KUKA KRL data list: C3_getcube.dat

&ACCESS RVO
&REL 4
&PARAM DISKPATH = KRC:\R1\Program
DEFDAT  C3_getcube PUBLIC

DECL E6POS XP1={X 224.960861,Y 55.9276581,Z 35.7754402,A 162.906586,B 89.0492325,C -106.826286,S 2,T 10,E1 0.0,E2 0.0,E3 0.0,E4 0.0,E5 0.0,E6 0.0}
DECL FDAT FP1={TOOL_NO 14,BASE_NO 2,IPO_FRAME #BASE,POINT2[] " ",TQ_STATE FALSE}
DECL PDAT PPDAT1={VEL 100.000,ACC 100.000,APO_DIST 100.000,GEAR_JERK 50.0000,EXAX_IGN 0}


ENDDAT
